TEXTLIST TL_SingleCylinderState
  0 = 'Uninitialized'
  10 = 'Initializing'
  20 = 'Ready initialized'
  30 = 'Idle'
  40 = 'Go active'
  50 = 'Go active done'
  60 = 'Go home'
  70 = 'Go home done'
  80 = 'Release'
  90 = 'Release done'
  100 = 'Reset'
  110 = 'Reset done'
  -10 = 'Aborting'
   = ''
END_TEXTLIST

(* stored: Version 1.1.0.1, ProductVersion 3.1.4024.12
   TextList TL_SingleCylinderState: Id {af5f9372-9ee5-4ef4-9e7c-b31a3c8df419} *)
